FUNCTION_BLOCK FB_Machine
VAR_INPUT
	
END_VAR
VAR_OUTPUT
END_VAR
VAR
	// =============== Common variables =========================================================
	bInit								: BOOL;									// True if module parameters are initialized	

		
	
	// =============== Machine elements =========================================================
	// This can be either Submodules or SubSystems
	fbMPG 			: 		FB_MPG ;		//MPG unit
	
	
	
	eMPGState : (INIT_START, WAIT_START, RUNNING);
	
	
	// =============== Testing ==================================================================
	_UINT : UINT;
	
	
END_VAR

// =========================================================
// Call of actions

	// Init
	General_Init();

	// Mode and state requests
	//General_Requests();
	
	// Enable for power supply, compressed air control and buttons
	//General_Enable();
	
	// Input variables of separating and sorting modules
	//General_ModuleInputs();
	
	// Output variables
	//General_SetOutput();
	
	// State machine
	//General_StateMachine();
	
	// Visualization
	//General_Visu();

// =========================================================
//TESTING


	_UINT := fbMPG.Value;

METHOD PRIVATE General_Init
VAR_INPUT
		
END_VAR
// =========================================================

IF NOT bInit THEN
	

	// Init done
		bInit := TRUE;
END_IF

// =========================================================
END_METHOD

METHOD General_StateMachine
VAR_INPUT
END_VAR
END_METHOD

METHOD PRIVATE Operating_Automatic
VAR_INPUT
END_VAR
END_METHOD

METHOD PRIVATE Operating_Manual
VAR_INPUT
END_VAR
END_METHOD

END_FUNCTION_BLOCK

(* stored: Version 1.1.0.1, ProductVersion 3.1.4024.11
   POU FB_Machine: Id {c1a5a3bc-1c08-4094-8c19-19b890488e0c}, SpecialFunc None
   Method General_Init: Id {f8d011be-fc17-4815-a997-af47d5450e1b}
   Method General_StateMachine: Id {49e44fbd-ba5a-4087-a8a2-9cb01d5be7ca}
   Method Operating_Automatic: Id {714f1efb-65b0-4136-9af7-6fcce3bba863}
   Method Operating_Manual: Id {b6a3ff7a-35ae-4a59-b2d8-519fd3fb4dfd} *)
